FUNCTION_BLOCK FB_GripperCtrl
VAR_INPUT
	
	bCloseGrip					:BOOL;
	bClosedSensor				:BOOL;

END_VAR
VAR_OUTPUT
	
	bOpen_Sig					:BOOL;
	bClose_Sig					:BOOL;
	bTimeout					:BOOL;

END_VAR
VAR
	tonOpenPulse				:Tc2_Standard.TON:=(PT:=T#1S);
	tonClosePulse				:Tc2_Standard.TON:=(PT:=T#1S);
	tonResetSignal				:ARRAY [1..2] OF Tc2_Standard.TON;
	tonTimeout					:Tc2_Standard.TON:=(PT:=T#3S);
	
END_VAR
//-------------------------------------------------------------------oldschoo1

//Timers
		 tonOpenPulse (IN:= NOT bCloseGrip);
		tonClosePulse (IN:= bCloseGrip);
		
	tonResetSignal[1] (IN:= NOT bCloseGrip,PT:=T#100MS);
	tonResetSignal[2] (IN:= bCloseGrip,PT:=T#100MS);
	
		   tonTimeout (IN:= bClose_Sig AND NOT bClosedSensor);

// Logic
IF NOT bCloseGrip THEN //-----------------------------------------------KEEP_OPEN

								bClose_Sig 		:= FALSE;
						
						IF tonResetSignal[1].Q 
							THEN	
								bOpen_Sig 		:= TRUE;
						END_IF							
ELSE //----------------------------------------------------------------CLOSE_GRIP
	
								bOpen_Sig 		:= FALSE;
						
							IF tonResetSignal[2].Q 
							THEN	
								bClose_Sig 		:= TRUE;
						END_IF										
END_IF
bTimeout := tonTimeout.Q; //----------------------------------------------TIMEOUT

//-----------------------------------------------------------------------oldschoo1

END_FUNCTION_BLOCK

(* stored: Version 1.1.0.1, ProductVersion 3.1.4024.12
   POU FB_GripperCtrl: Id {8d7a70bf-818b-4d26-bc5f-665d377e6ae1}, SpecialFunc None *)
